# EPICS autosave request: apps/chillerApp/Db/presto_settings.req
#
# Presto Temperature Control System - Models A80(t), W80(t)
#
# Author: Wesley Moore
# Date:   Jan 2015
#

$(P)$(R)TEMP:SP
$(P)$(R)PUMP_PRES:SP
